{attribute 'qualified_only'}
{attribute 'strict'}
TYPE E_Gen24_ChargeState :
(
	eNoDataReceived := 0,
	eOff := 1,
	eEmpty := 2,
	eDischarge := 3,
	eCharging := 4,
	eFull := 5,
	eHolding := 6,
	eTesting := 7
);
END_TYPE

(* stored: Version 1.1.0.1, ProductVersion 3.1.4024.6
   DUT E_Gen24_ChargeState: Id {b9ada85e-9894-4069-81eb-17ac145024f4} *)
